(* Schneider Machine Expert - Basic project Trafficlights V2, file version 2.6.0.0 *)
(* ProjectInformations: Name=New project *)

HARDWARE
  Cpu 0: TM221CE16R
  EthernetConfiguration: NetworkName=M221, IpAllocationMode=FixedAddress, IpAddress=192.168.1.3, SubnetMask=255.255.255.0
  SerialLineConfiguration: Baud=Baud19200, Parity=ParityEven, DataBits=DataBits8, StopBits=StopBits1, PhysicalMedium=PhysicalMediumRs485, TransmissionMode=TransmissionModeModbusRtu, SlaveId=1, Addressing=SlaveAddressing
  MastTask: UsePeriodScanMode=false, PeriodScan=100
  FastTask: Period=255
  CpuBehavior: StartingMode=StartAsPreviousState, AutoSaveRamOnEeprom=true, WatchdogPeriod=250

SYMBOLS  (address, symbol, comment, settings)
  %M0       STV1
  %M1       STV2
  %M3       STV3
  %M4       STV4
  %M6       MEM
  %M10      FIRST_TIME
  %M15      START_PR
  %MW1      CODW1
  %MW2      CODW2
  %MW4      TEMP1
  %MW5      TEMP2
  %MW6      MEM1
  %MW7      MEM2
  %MW8      MEM3
  %MW9      MEM4
  %MW11     TIME_GR
  %MW12     TIME_YE
  %MW13     TIME_RE
  %TM0      RED_LIGHT  [Type=TP, Preset=21, Base=OneSecond]
  %TM1      GREEN_LIGHT  [Type=TP, Preset=8, Base=OneSecond]
  %TM2      YELLOW_LIGHT  [Type=TP, Preset=4, Base=OneSecond]
  %TM3      TOSTART  [Type=TP, Preset=8, Base=OneSecond]
  %I0.0     SET1
  %I0.3     SET3
  %Q0.0     OUT1
  %Q0.1     OUT2

POU New POU
  (* SectionNumber=1 *)

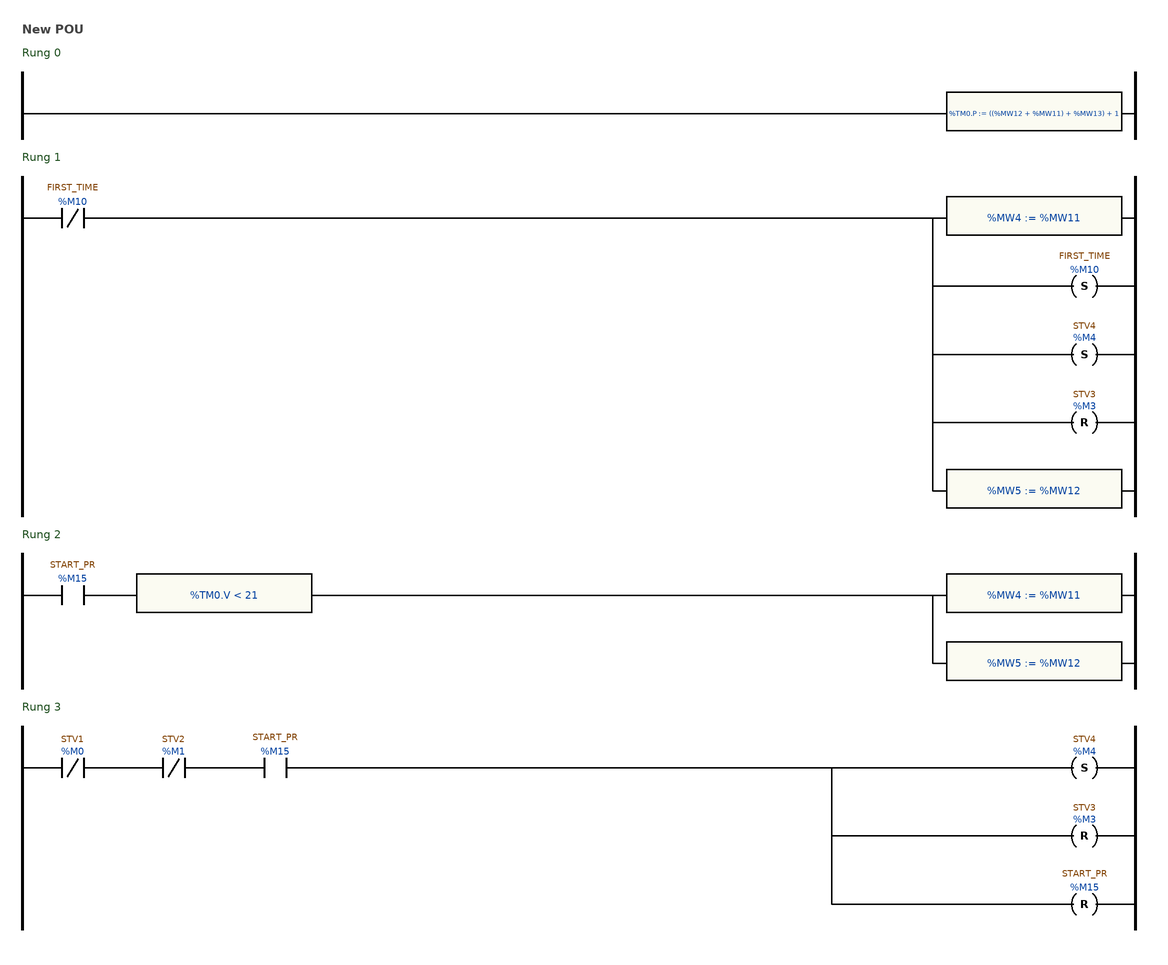

// Rung 0
  LD 1
  [ %TM0.P := ( ( %MW12 + %MW11 ) + %MW13 ) + 1 ](* RED_LIGHT, TIME_YE, TIME_GR, TIME_RE *)
  // as ST:
  //   RED_LIGHT.P := ( ( TIME_YE + TIME_GR ) + TIME_RE ) + 1;

// Rung 1
  LDN %M10                (* FIRST_TIME *)
  [ %MW4 := %MW11 ]       (* TEMP1, TIME_GR *)
  S %M10                  (* FIRST_TIME *)
  S %M4                   (* STV4 *)
  R %M3                   (* STV3 *)
  [ %MW5 := %MW12 ]       (* TEMP2, TIME_YE *)
  // as ST:
  //   IF NOT FIRST_TIME THEN TEMP1 := TIME_GR; END_IF;
  //   _t1 := NOT FIRST_TIME;
  //   IF _t1 THEN FIRST_TIME := TRUE; END_IF;
  //   IF _t1 THEN STV4 := TRUE; END_IF;
  //   IF _t1 THEN STV3 := FALSE; END_IF;
  //   IF _t1 THEN TEMP2 := TIME_YE; END_IF;

// Rung 2
  LD %M15                 (* START_PR *)
  AND [ %TM0.V < 21 ]     (* RED_LIGHT *)
  [ %MW4 := %MW11 ]       (* TEMP1, TIME_GR *)
  [ %MW5 := %MW12 ]       (* TEMP2, TIME_YE *)
  // as ST:
  //   IF START_PR AND RED_LIGHT.V < 21 THEN TEMP1 := TIME_GR; END_IF;
  //   IF START_PR AND RED_LIGHT.V < 21 THEN TEMP2 := TIME_YE; END_IF;

// Rung 3
  LDN %M0                 (* STV1 *)
  ANDN %M1                (* STV2 *)
  AND %M15                (* START_PR *)
  S %M4                   (* STV4 *)
  R %M3                   (* STV3 *)
  R %M15                  (* START_PR *)
  // as ST:
  //   IF NOT STV1 AND NOT STV2 AND START_PR THEN STV4 := TRUE; END_IF;
  //   IF NOT STV1 AND NOT STV2 AND START_PR THEN STV3 := FALSE; END_IF;
  //   IF NOT STV1 AND NOT STV2 AND START_PR THEN START_PR := FALSE; END_IF;

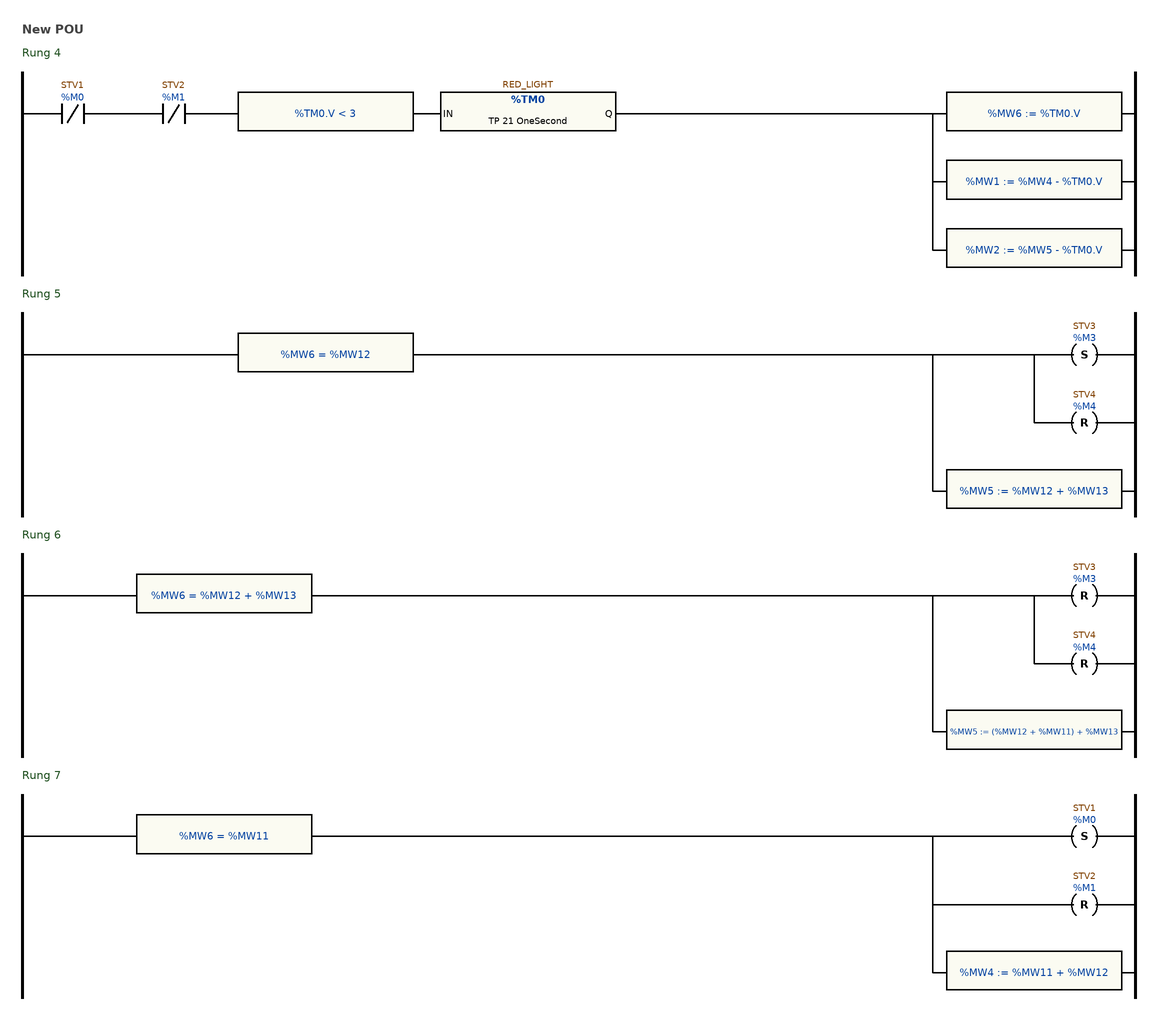

// Rung 4
  BLK %TM0                (* RED_LIGHT *)
  LDN %M0                 (* STV1 *)
  ANDN %M1                (* STV2 *)
  AND [ %TM0.V < 3 ]      (* RED_LIGHT *)
  IN
  OUT_BLK
  LD Q
  [ %MW6 := %TM0.V ]      (* MEM1, RED_LIGHT *)
  [ %MW1 := %MW4 - %TM0.V ](* CODW1, TEMP1, RED_LIGHT *)
  [ %MW2 := %MW5 - %TM0.V ](* CODW2, TEMP2, RED_LIGHT *)
  END_BLK
  // as ST:
  //   RED_LIGHT(IN := NOT STV1 AND NOT STV2 AND RED_LIGHT.V < 3);
  //   IF RED_LIGHT.Q THEN MEM1 := RED_LIGHT.V; END_IF;
  //   IF RED_LIGHT.Q THEN CODW1 := TEMP1 - RED_LIGHT.V; END_IF;
  //   IF RED_LIGHT.Q THEN CODW2 := TEMP2 - RED_LIGHT.V; END_IF;

// Rung 5
  LD [ %MW6 = %MW12 ]     (* MEM1, TIME_YE *)
  S %M3                   (* STV3 *)
  R %M4                   (* STV4 *)
  [ %MW5 := %MW12 + %MW13 ](* TEMP2, TIME_YE, TIME_RE *)
  // as ST:
  //   IF MEM1 = TIME_YE THEN STV3 := TRUE; END_IF;
  //   IF MEM1 = TIME_YE THEN STV4 := FALSE; END_IF;
  //   IF MEM1 = TIME_YE THEN TEMP2 := TIME_YE + TIME_RE; END_IF;

// Rung 6
  LD 1
  AND [ %MW6 = %MW12 + %MW13 ](* MEM1, TIME_YE, TIME_RE *)
  R %M3                   (* STV3 *)
  R %M4                   (* STV4 *)
  [ %MW5 := ( %MW12 + %MW11 ) + %MW13 ](* TEMP2, TIME_YE, TIME_GR, TIME_RE *)
  // as ST:
  //   IF MEM1 = TIME_YE + TIME_RE THEN STV3 := FALSE; END_IF;
  //   IF MEM1 = TIME_YE + TIME_RE THEN STV4 := FALSE; END_IF;
  //   IF MEM1 = TIME_YE + TIME_RE THEN TEMP2 := ( TIME_YE + TIME_GR ) + TIME_RE; END_IF;

// Rung 7
  LD [ %MW6 = %MW11 ]     (* MEM1, TIME_GR *)
  S %M0                   (* STV1 *)
  R %M1                   (* STV2 *)
  [ %MW4 := %MW11 + %MW12 ](* TEMP1, TIME_GR, TIME_YE *)
  // as ST:
  //   IF MEM1 = TIME_GR THEN STV1 := TRUE; END_IF;
  //   IF MEM1 = TIME_GR THEN STV2 := FALSE; END_IF;
  //   IF MEM1 = TIME_GR THEN TEMP1 := TIME_GR + TIME_YE; END_IF;

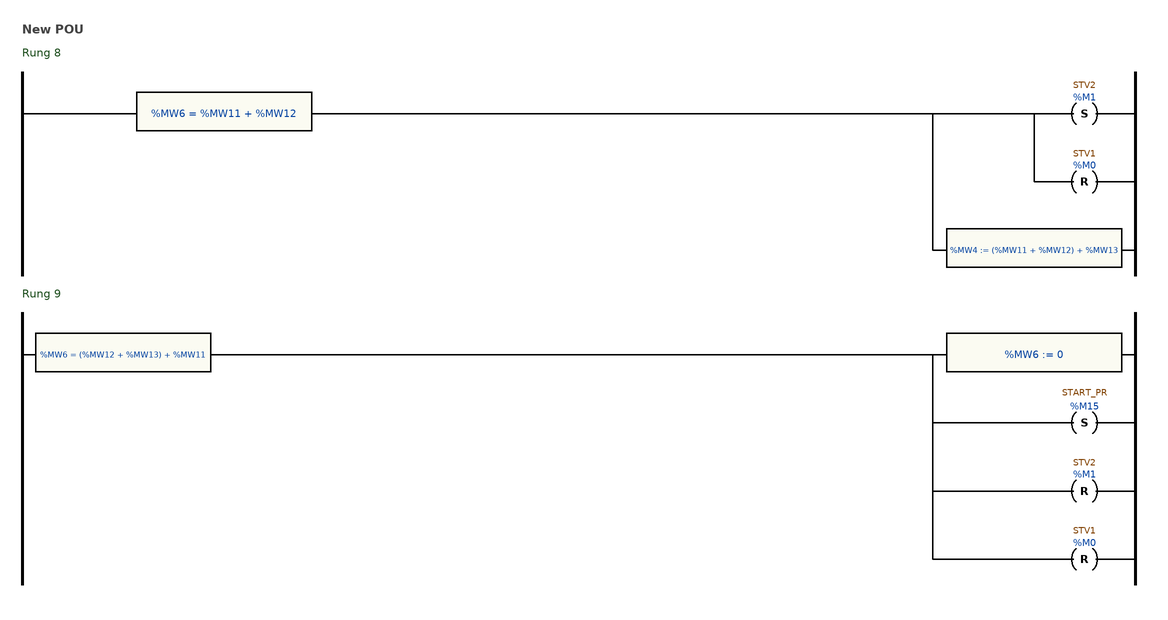

// Rung 8
  LD 1
  AND [ %MW6 = %MW11 + %MW12 ](* MEM1, TIME_GR, TIME_YE *)
  S %M1                   (* STV2 *)
  R %M0                   (* STV1 *)
  [ %MW4 := ( %MW11 + %MW12 ) + %MW13 ](* TEMP1, TIME_GR, TIME_YE, TIME_RE *)
  // as ST:
  //   IF MEM1 = TIME_GR + TIME_YE THEN STV2 := TRUE; END_IF;
  //   IF MEM1 = TIME_GR + TIME_YE THEN STV1 := FALSE; END_IF;
  //   IF MEM1 = TIME_GR + TIME_YE THEN TEMP1 := ( TIME_GR + TIME_YE ) + TIME_RE; END_IF;

// Rung 9
  LD 1
  AND [ %MW6 = ( %MW12 + %MW13 ) + %MW11 ](* MEM1, TIME_YE, TIME_RE, TIME_GR *)
  [ %MW6 := 0 ]           (* MEM1 *)
  S %M15                  (* START_PR *)
  R %M1                   (* STV2 *)
  R %M0                   (* STV1 *)
  // as ST:
  //   _t1 := MEM1 = ( TIME_YE + TIME_RE ) + TIME_GR;
  //   IF _t1 THEN MEM1 := 0; END_IF;
  //   IF _t1 THEN START_PR := TRUE; END_IF;
  //   IF _t1 THEN STV2 := FALSE; END_IF;
  //   IF _t1 THEN STV1 := FALSE; END_IF;
